{attribute 'qualified_only'}
VAR_GLOBAL
	inputl   AT%I*   :BOOL;
	output2  AT%Q*  :BOOL;
	JoinTrack: INT;
	
	bBusyA:BOOL;
	bBusyB:BOOL;
	bDoneA:BOOL;
	bDoneB:BOOL;
	bfill:BOOL;
	bstop:BOOL;

END_VAR

VAR_GLOBAL CONSTANT
	MAX_MOVER     :INT:=3; //0 to...
	MAX_FEEDBACK  :INT:=100;
	MAX_Track     :INT:=7;
END_VAR

(* stored: Version 1.1.0.1
   GVL GVL: Id {59c74646-7473-42d8-b33e-cdd2bd3b98de} *)
